// TIA Portal project "Smart-greenhouse" (V16)

(* hardware
DEVICE "S7-1200 station_1"  S7-1200 Station
   slot 0: "Telaio di montaggio_0"  S7-1200 Rack  Rack  V1.0
   slot 1: "PLC_1"  CPU 1212C AC/DC/Rly  6ES7 212-1BE40-0XB0  V4.4
*)

// ===== PLC "PLC_1"  CPU 1212C AC/DC/Rly =====

VAR_GLOBAL   // PLC tag table "Tabella delle variabili standard"
   "GripperOpenStop" AT %I0.0 : Bool;
   "GripperCounter" AT %I0.1 : Bool;
   "ArmBackStop" AT %I0.2 : Bool;
   "ArmHCounter" AT %I0.3 : Bool;
   "ArmTopStop" AT %I0.4 : Bool;
   "ArmRotationStop" AT %I0.5 : Bool;
   "RotationalEncoder" AT %ID1000 : DInt;
   "VerticalEncoder" AT %ID1004 : DInt;
   "ConnectionButton" AT %I1.2 : Bool;
   "StopButton" AT %I1.3 : Bool;
   "ResetButton" AT %I1.4 : Bool;
   "Photosensor" AT %I1.5 : Bool;
   "GripperOpen" AT %Q0.0 : Bool;
   "GripperClose" AT %Q0.1 : Bool;
   "ArmFront" AT %Q0.2 : Bool;
   "ArmBack" AT %Q0.3 : Bool;
   "ArmDown" AT %Q0.4 : Bool;
   "ArmUp" AT %Q0.5 : Bool;
   "RotationClockwise" AT %Q0.6 : Bool;
   "RotationCounterclockwise" AT %Q0.7 : Bool;
   "GreenLed" AT %Q1.0 : Bool;
   "StopConveyor" AT %Q1.1 : Bool;
   "System_Byte" AT %MB1 : Byte;
   "FirstScan" AT %M6.0 : Bool;
   "DiagStatusUpdate" AT %M6.1 : Bool;
   "AlwaysTRUE" AT %M6.2 : Bool;
   "AlwaysFALSE" AT %M6.3 : Bool;
   "RotationalCounter" AT %MW2 : UInt;
   "Clock_Byte" AT %MB0 : Byte;
   "Clock_10Hz" AT %M0.0 : Bool;
   "Clock_5Hz" AT %M0.1 : Bool;
   "Clock_2.5Hz" AT %M0.2 : Bool;
   "Clock_2Hz" AT %M0.3 : Bool;
   "Clock_1.25Hz" AT %M0.4 : Bool;
   "Clock_1Hz" AT %M0.5 : Bool;
   "Clock_0.625Hz" AT %M0.6 : Bool;
   "Clock_0.5Hz" AT %M0.7 : Bool;
   "VerticalCounter" AT %MW4 : UInt;
   "ForceReset" AT %M7.0 : Bool;
   "ResetCompleted" AT %M7.1 : Bool;
   "TCON_Req" AT %M1.0 : Bool;
   "TDIS_Req" AT %M1.1 : Bool;
   "TSEND_Req" AT %M1.2 : Bool;
   "TRCV_Req" AT %M1.3 : Bool;
   "VerticalOverCounter" AT %MW8 : Int;
   "VerticalUnderCounter" AT %MW10 : Int;
   "RotationOverCounter" AT %MW12 : Int;
   "RotationUnderCounter" AT %MW14 : Int;
   "NormalizedRotationUnderCounter" AT %MW16 : Int;
   "NormalizedVerticalUnderCounter" AT %MW18 : Int;
   "StopAll" AT %M20.1 : Bool;
   "HRegistered" AT %M20.2 : Bool;
   "RRegistered" AT %M20.3 : Bool;
   "VRegistered" AT %M20.4 : Bool;
   "State 0" AT %M20.5 : Bool;
   "State 3" AT %M20.6 : Bool;
   "AuxPhotocellStatus" AT %M20.7 : Bool;
   "State 3.1" AT %M21.0 : Bool;
   "State 3.2" AT %M21.1 : Bool;
   "HallEffectSensor" AT %I1.6 : Bool;
   "Sprinkler" AT %Q1.2 : Bool;
   "ArmTriggerOut_REQ" AT %M21.2 : Bool;
   "Test" AT %M21.3 : Bool;
   "MotorOn" AT %M21.4 : Bool;
   "TESTSOCKET" AT %M21.5 : Bool;
   "ForceMotor" AT %M21.6 : Bool;
   "AuxStop" AT %M21.7 : Bool;
   "State 3.1.1" AT %M22.0 : Bool;
   "State 3.1.2" AT %M22.1 : Bool;
   "State 3.1.3" AT %M22.2 : Bool;
   "State 3.3" AT %M22.3 : Bool;
   "State 1" AT %M22.4 : Bool;
   "State 1.1" AT %M22.5 : Bool;
   "State 1.2" AT %M22.6 : Bool;
   "State 1.3" AT %M22.7 : Bool;
   "State 2" AT %M23.0 : Bool;
   "AuxLapNotCompleted" AT %M23.1 : Bool;
   "HighTemp" AT %I1.7 : Bool;
   "LowTemp" AT %I2.0 : Bool;
   "HighHum" AT %I2.1 : Bool;
   "AuxHighTemp" AT %M23.2 : Bool;
   "AuxLowTemp" AT %M23.3 : Bool;
   "AuxHum" AT %M23.4 : Bool;
   "WindowPiston" AT %Q1.3 : Bool;
   "IRLamp" AT %Q1.4 : Bool;
   "Fan" AT %Q1.5 : Bool;
   "Tag_1" AT %MW0 : Int;
END_VAR

DATA_BLOCK "REAL TIME DATA"   // DB4
{ S7_Optimized_Access := 'TRUE' }
VERSION : 0.1
   VAR
      "REAL TIME DATA" : DTL;
   END_VAR
BEGIN
END_DATA_BLOCK

DATA_BLOCK "Trigger_values"   // DB7
{ S7_Optimized_Access := 'FALSE' }
VERSION : 0.1
   VAR
      Trigger : Bool;
   END_VAR
BEGIN
END_DATA_BLOCK

DATA_BLOCK "Sent_values"   // DB10
{ S7_Optimized_Access := 'FALSE' }
VERSION : 0.1
   VAR
      Rotation : Int;
      Vertical : Int;
      Horizontal : Int;
      Gripper : Bool;
   END_VAR
BEGIN
END_DATA_BLOCK

DATA_BLOCK "Received_values"   // DB12
{ S7_Optimized_Access := 'FALSE' }
VERSION : 0.1
   VAR
      Rotation : Int;
      Vertical : Int;
      Horizontal : Int;
      Gripper : Bool;
   END_VAR
BEGIN
END_DATA_BLOCK

DATA_BLOCK "Obj_detect"   // DB20
{ S7_Optimized_Access := 'FALSE' }
VERSION : 0.1
   VAR
      message : String := 'START';
   END_VAR
BEGIN
END_DATA_BLOCK

// folder: System blocks/Program resources

DATA_BLOCK "CONTATORE"   // DB1
{ S7_Optimized_Access := 'TRUE' }
AUTHOR : Simatic
FAMILY : IEC
NAME : CNTR
VERSION : 1.0
// stored: InstanceOfName IEC_COUNTER
"IEC_COUNTER"
BEGIN
END_DATA_BLOCK

DATA_BLOCK "Timer Sprinkler"   // DB2
{ S7_Optimized_Access := 'TRUE' }
AUTHOR : Simatic
FAMILY : IEC
NAME : IEC_TMR
VERSION : 1.0
// stored: InstanceOfName IEC_TIMER
"IEC_TIMER"
BEGIN
END_DATA_BLOCK

DATA_BLOCK "ArmHCounterCTUD"   // DB3
{ S7_Optimized_Access := 'TRUE' }
AUTHOR : Simatic
FAMILY : IEC
NAME : CNTR
VERSION : 1.0
// stored: InstanceOfName IEC_COUNTER
"IEC_COUNTER"
BEGIN
END_DATA_BLOCK

DATA_BLOCK "PLC_1_Connection_DB"   // DB6
{ S7_Optimized_Access := 'TRUE' }
AUTHOR : SIMATIC
FAMILY : MC7Plus
NAME : TC_IP_v4
VERSION : 1.0
// stored: InstanceOfName TCON_IP_v4
"TCON_IP_v4"
BEGIN
   ID := 1;
   InterfaceId := 64;
   RemotePort := 2001;
   ActiveEstablished := true;
   RemoteAddress.ADDR[1] := 192;
   RemoteAddress.ADDR[2] := 168;
   RemoteAddress.ADDR[4] := 9;
END_DATA_BLOCK

DATA_BLOCK "ArmHStatusCTUD"   // DB9
{ S7_Optimized_Access := 'TRUE' }
AUTHOR : Simatic
FAMILY : IEC
NAME : CNTR
VERSION : 1.0
// stored: InstanceOfName IEC_COUNTER
"IEC_COUNTER"
BEGIN
END_DATA_BLOCK

DATA_BLOCK "GripperStatus"   // DB15
{ S7_Optimized_Access := 'TRUE' }
AUTHOR : Simatic
FAMILY : IEC
NAME : CNTR
VERSION : 1.0
// stored: InstanceOfName IEC_COUNTER
"IEC_COUNTER"
BEGIN
END_DATA_BLOCK

DATA_BLOCK "ArmHStatus"   // DB16
{ S7_Optimized_Access := 'TRUE' }
AUTHOR : Simatic
FAMILY : IEC
NAME : CNTR
VERSION : 1.0
// stored: InstanceOfName IEC_COUNTER
"IEC_COUNTER"
BEGIN
END_DATA_BLOCK

DATA_BLOCK "IEC_Timer_0_DB"   // DB17
{ S7_Optimized_Access := 'TRUE' }
AUTHOR : Simatic
FAMILY : IEC
NAME : IEC_TMR
VERSION : 1.0
// stored: InstanceOfName IEC_TIMER
"IEC_TIMER"
BEGIN
END_DATA_BLOCK

DATA_BLOCK "IEC_Timer_0_DB_1"   // DB18
{ S7_Optimized_Access := 'TRUE' }
AUTHOR : Simatic
FAMILY : IEC
NAME : IEC_TMR
VERSION : 1.0
// stored: InstanceOfName IEC_TIMER
"IEC_TIMER"
BEGIN
END_DATA_BLOCK

// folder: (top level)

ORGANIZATION_BLOCK "Main"   // OB1, LAD, ProgramCycle
TITLE = "Main Program Sweep (Cycle)"
{ S7_Optimized_Access := 'TRUE' }
VERSION : 0.1
   VAR_INPUT
      Initial_Call : Bool;   // Initial call of this OB
      Remanence : Bool;   // =True, if remanent data are available
   END_VAR
   VAR_TEMP   // added for the SCL form of the ladder/FBD networks
      _w1 : Bool;
      _w2 : Bool;
      _w3 : Bool;
      _w4 : Bool;
      _w5 : Bool;
      _w6 : Bool;
      _w7 : Bool;
   END_VAR
BEGIN

REGION Network 1: State inizialization
   // All'avvio del PLC vengono inizializzati gli stati
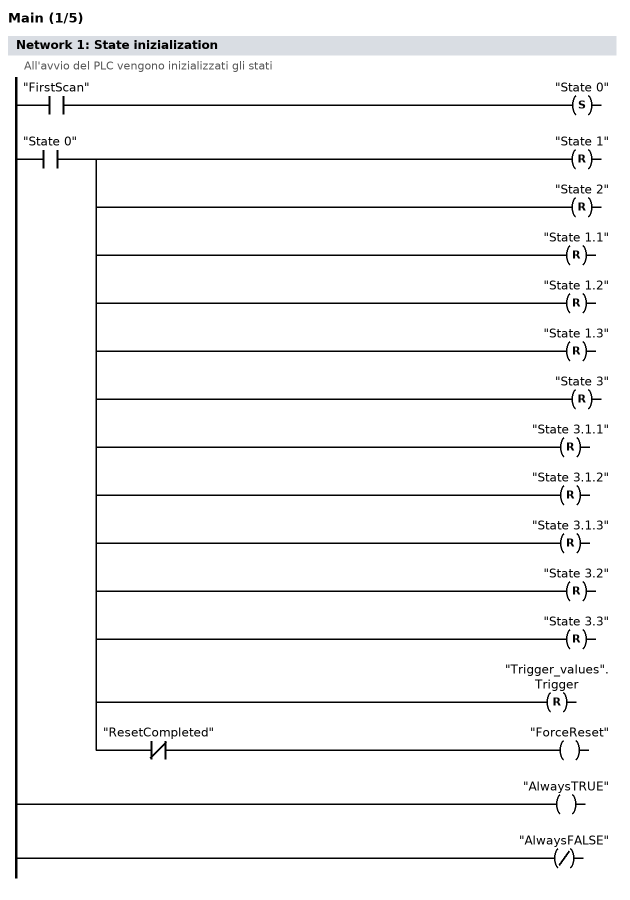
   RUNG wire#powerrail
      Contact( "FirstScan" )
      S_Coil( "State 0" )
   END_RUNG
   RUNG wire#powerrail
      Contact( "State 0" )
      wire#w1
      R_Coil( "State 1" )
   END_RUNG
   RUNG wire#w1
      R_Coil( "State 2" )
   END_RUNG
   RUNG wire#w1
      R_Coil( "State 1.1" )
   END_RUNG
   RUNG wire#w1
      R_Coil( "State 1.2" )
   END_RUNG
   RUNG wire#w1
      R_Coil( "State 1.3" )
   END_RUNG
   RUNG wire#w1
      R_Coil( "State 3" )
   END_RUNG
   RUNG wire#w1
      R_Coil( "State 3.1.1" )
   END_RUNG
   RUNG wire#w1
      R_Coil( "State 3.1.2" )
   END_RUNG
   RUNG wire#w1
      R_Coil( "State 3.1.3" )
   END_RUNG
   RUNG wire#w1
      R_Coil( "State 3.2" )
   END_RUNG
   RUNG wire#w1
      R_Coil( "State 3.3" )
   END_RUNG
   RUNG wire#w1
      R_Coil( "Trigger_values".Trigger )
   END_RUNG
   RUNG wire#w1
      I_Contact( "ResetCompleted" )
      Coil( "ForceReset" )
   END_RUNG
   RUNG wire#powerrail
      Coil( "AlwaysTRUE" )
   END_RUNG
   RUNG wire#powerrail
      I_Coil( "AlwaysFALSE" )
   END_RUNG
   // the same network as SCL:
   IF "FirstScan" THEN "State 0" := TRUE; END_IF;
   IF "State 0" THEN
       "State 1" := FALSE;
       "State 2" := FALSE;
       "State 1.1" := FALSE;
       "State 1.2" := FALSE;
       "State 1.3" := FALSE;
       "State 3" := FALSE;
       "State 3.1.1" := FALSE;
       "State 3.1.2" := FALSE;
       "State 3.1.3" := FALSE;
       "State 3.2" := FALSE;
       "State 3.3" := FALSE;
       "Trigger_values".Trigger := FALSE;
   END_IF;
   "ForceReset" := "State 0" AND NOT "ResetCompleted";
   "AlwaysTRUE" := TRUE;
   "AlwaysFALSE" := NOT TRUE;
END_REGION

REGION Network 2: Gestione braccio robotico
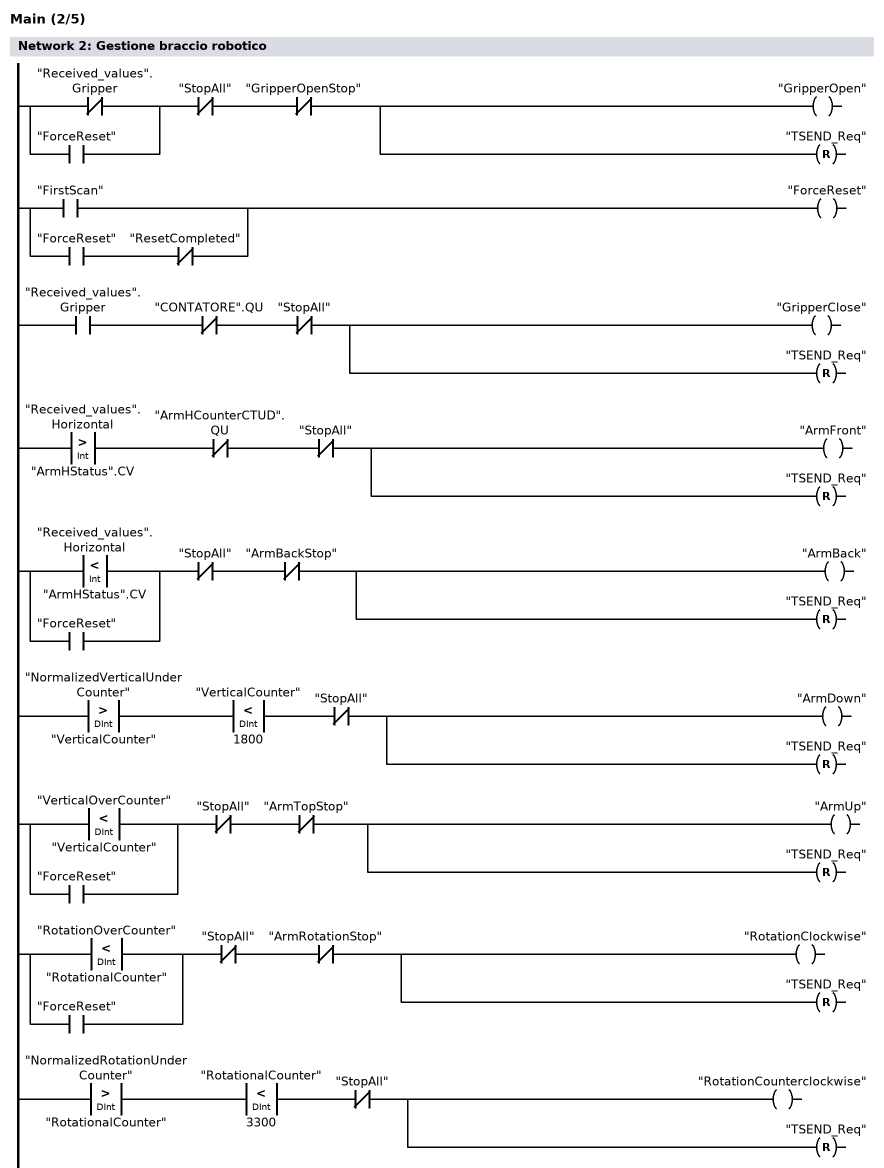
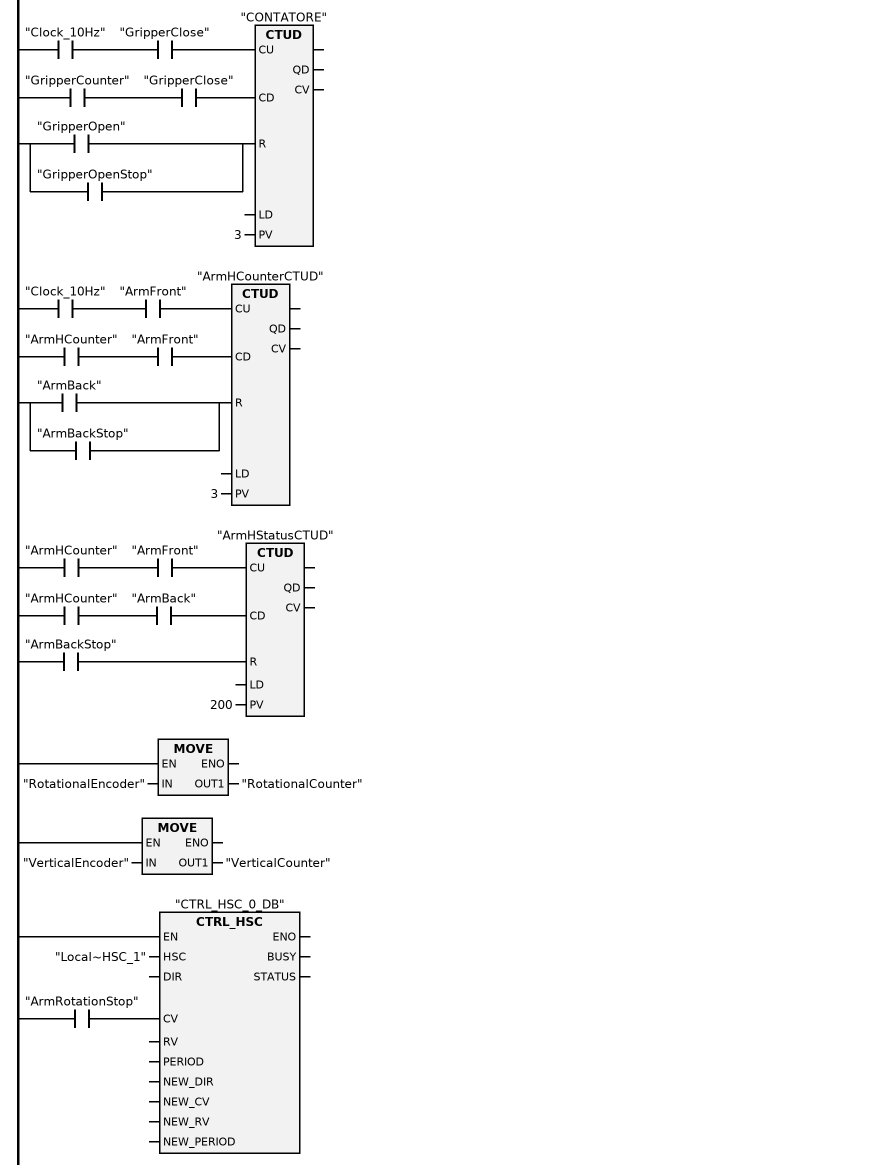
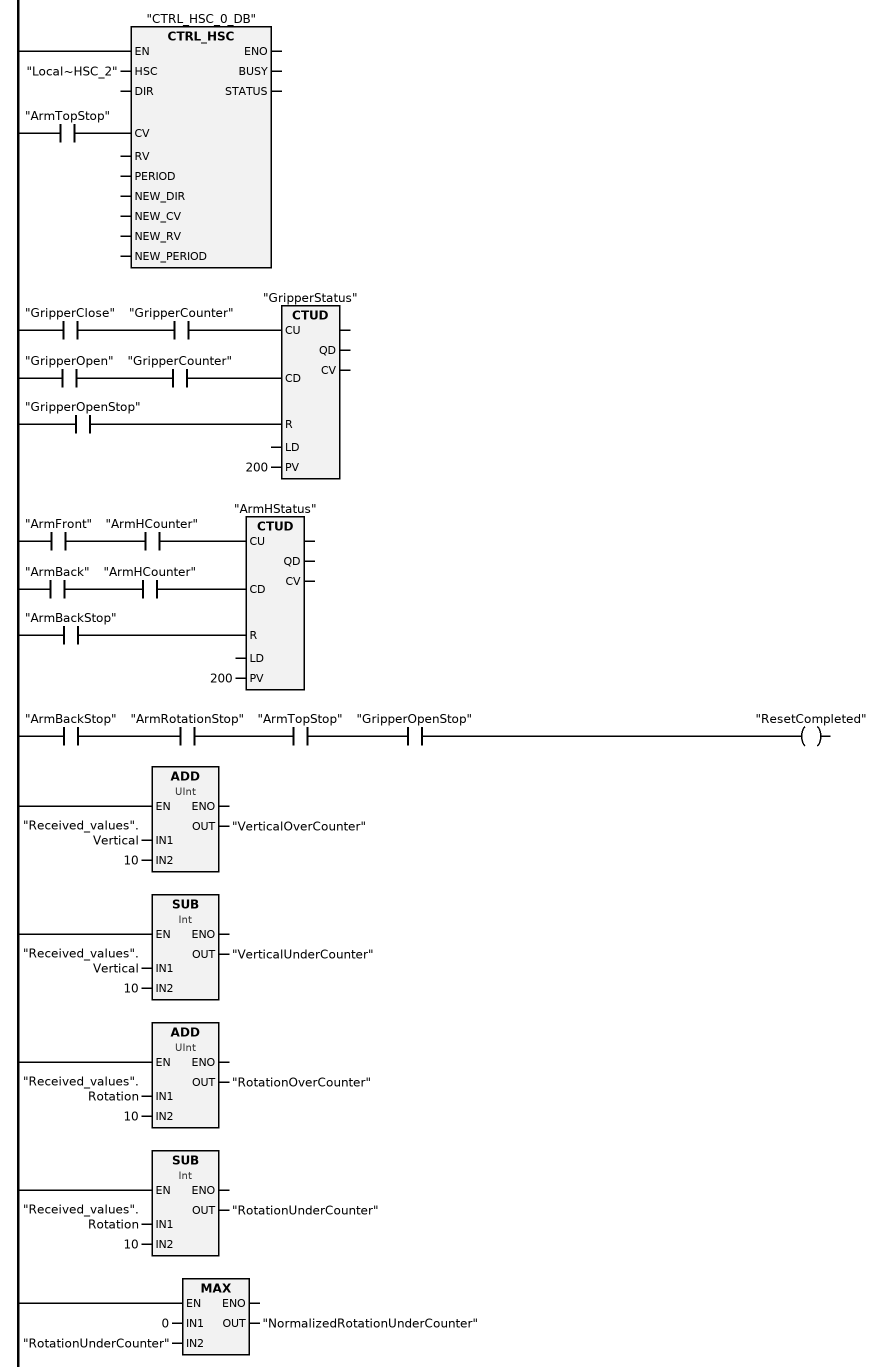
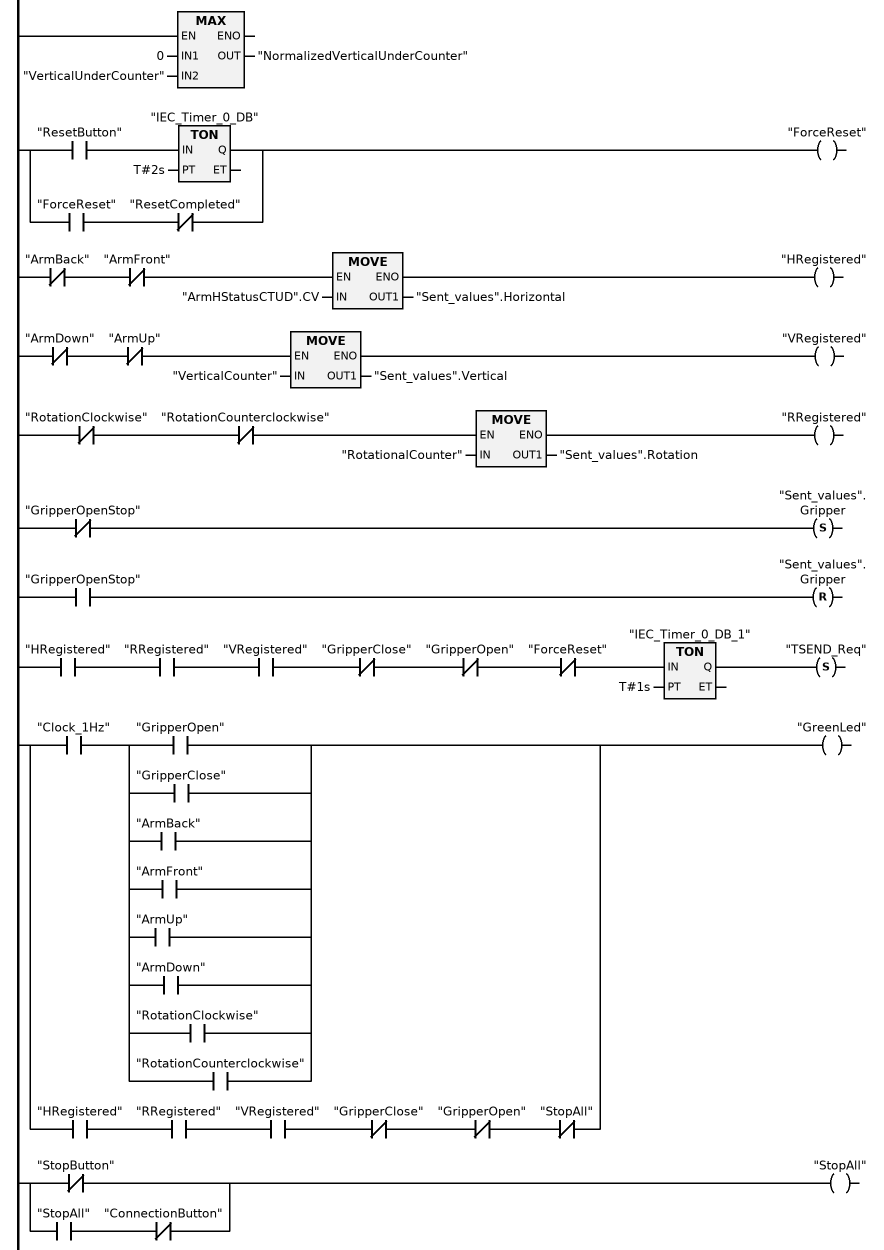
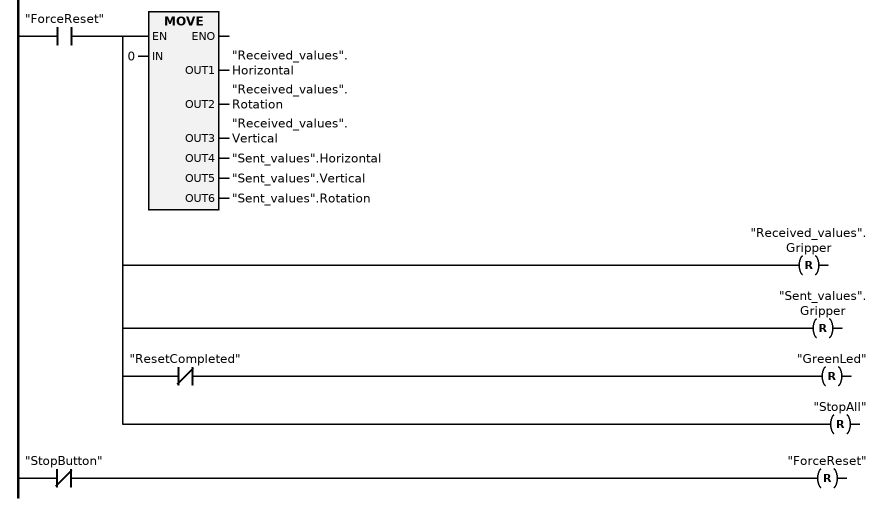
   "GripperOpen" := (NOT "Received_values".Gripper OR "ForceReset") AND NOT "StopAll" AND NOT "GripperOpenStop";
   IF "GripperOpen" THEN "TSEND_Req" := FALSE; END_IF;
   "ForceReset" := "FirstScan" OR ("ForceReset" AND NOT "ResetCompleted");
   "GripperClose" := "Received_values".Gripper AND NOT "CONTATORE".QU AND NOT "StopAll";
   IF "GripperClose" THEN "TSEND_Req" := FALSE; END_IF;
   "ArmFront" := ("Received_values".Horizontal > "ArmHStatus".CV) AND NOT "ArmHCounterCTUD".QU AND NOT "StopAll";
   IF "ArmFront" THEN "TSEND_Req" := FALSE; END_IF;
   "ArmBack" := (("Received_values".Horizontal < "ArmHStatus".CV) OR "ForceReset") AND NOT "StopAll" AND NOT "ArmBackStop";
   IF "ArmBack" THEN "TSEND_Req" := FALSE; END_IF;
   "ArmDown" := ("NormalizedVerticalUnderCounter" > "VerticalCounter") AND ("VerticalCounter" < 1800) AND NOT "StopAll";
   IF "ArmDown" THEN "TSEND_Req" := FALSE; END_IF;
   "ArmUp" := (("VerticalOverCounter" < "VerticalCounter") OR "ForceReset") AND NOT "StopAll" AND NOT "ArmTopStop";
   IF "ArmUp" THEN "TSEND_Req" := FALSE; END_IF;
   "RotationClockwise" := (("RotationOverCounter" < "RotationalCounter") OR "ForceReset") AND NOT "StopAll" AND NOT "ArmRotationStop";
   IF "RotationClockwise" THEN "TSEND_Req" := FALSE; END_IF;
   "RotationCounterclockwise" := ("NormalizedRotationUnderCounter" > "RotationalCounter") AND ("RotationalCounter" < 3300) AND NOT "StopAll";
   IF "RotationCounterclockwise" THEN "TSEND_Req" := FALSE; END_IF;
   "CONTATORE".CTUD(CU := "Clock_10Hz" AND "GripperClose",
                    CD := "GripperCounter" AND "GripperClose",
                    R := "GripperOpen" OR "GripperOpenStop",
                    PV := 3);
   "ArmHCounterCTUD".CTUD(CU := "Clock_10Hz" AND "ArmFront",
                          CD := "ArmHCounter" AND "ArmFront",
                          R := "ArmBack" OR "ArmBackStop",
                          PV := 3);
   "ArmHStatusCTUD".CTUD(CU := "ArmHCounter" AND "ArmFront",
                         CD := "ArmHCounter" AND "ArmBack",
                         R := "ArmBackStop",
                         PV := 200);
   "RotationalCounter" := "RotationalEncoder";
   "VerticalCounter" := "VerticalEncoder";
   "CTRL_HSC_0_DB"(HSC := "Local~HSC_1", CV := "ArmRotationStop");   // CTRL_HSC
   "CTRL_HSC_0_DB"(HSC := "Local~HSC_2", CV := "ArmTopStop");   // CTRL_HSC
   "GripperStatus".CTUD(CU := "GripperClose" AND "GripperCounter",
                        CD := "GripperOpen" AND "GripperCounter",
                        R := "GripperOpenStop",
                        PV := 200);
   "ArmHStatus".CTUD(CU := "ArmFront" AND "ArmHCounter",
                     CD := "ArmBack" AND "ArmHCounter",
                     R := "ArmBackStop",
                     PV := 200);
   "ResetCompleted" := "ArmBackStop" AND "ArmRotationStop" AND "ArmTopStop" AND "GripperOpenStop";
   "VerticalOverCounter" := "Received_values".Vertical + 10;
   "VerticalUnderCounter" := "Received_values".Vertical - 10;
   "RotationOverCounter" := "Received_values".Rotation + 10;
   "RotationUnderCounter" := "Received_values".Rotation - 10;
   "NormalizedRotationUnderCounter" := MAX(IN1 := 0, IN2 := "RotationUnderCounter");
   "NormalizedVerticalUnderCounter" := MAX(IN1 := 0, IN2 := "VerticalUnderCounter");
   "IEC_Timer_0_DB".TON(IN := "ResetButton", PT := T#2s);
   "ForceReset" := "IEC_Timer_0_DB".Q OR ("ForceReset" AND NOT "ResetCompleted");
   #_w1 := NOT "ArmBack" AND NOT "ArmFront";
   IF #_w1 THEN "Sent_values".Horizontal := "ArmHStatusCTUD".CV; END_IF;
   "HRegistered" := #_w1;
   #_w2 := NOT "ArmDown" AND NOT "ArmUp";
   IF #_w2 THEN "Sent_values".Vertical := "VerticalCounter"; END_IF;
   "VRegistered" := #_w2;
   #_w3 := NOT "RotationClockwise" AND NOT "RotationCounterclockwise";
   IF #_w3 THEN "Sent_values".Rotation := "RotationalCounter"; END_IF;
   "RRegistered" := #_w3;
   IF NOT "GripperOpenStop" THEN "Sent_values".Gripper := TRUE; END_IF;
   IF "GripperOpenStop" THEN "Sent_values".Gripper := FALSE; END_IF;
   "IEC_Timer_0_DB_1".TON(IN := "HRegistered" AND "RRegistered" AND "VRegistered" AND NOT "GripperClose" AND NOT "GripperOpen" AND NOT "ForceReset",
                          PT := T#1s);
   IF "IEC_Timer_0_DB_1".Q THEN "TSEND_Req" := TRUE; END_IF;
   "GreenLed" := ("Clock_1Hz" AND ("GripperOpen" OR "GripperClose" OR "ArmBack" OR "ArmFront" OR "ArmUp" OR "ArmDown" OR "RotationClockwise" OR "RotationCounterclockwise")) OR ("HRegistered" AND "RRegistered" AND "VRegistered" AND NOT "GripperClose" AND NOT "GripperOpen" AND NOT "StopAll");
   "StopAll" := NOT "StopButton" OR ("StopAll" AND NOT "ConnectionButton");
   IF "ForceReset" THEN
       "Received_values".Horizontal := 0;
       "Received_values".Rotation := 0;
       "Received_values".Vertical := 0;
       "Sent_values".Horizontal := 0;
       "Sent_values".Vertical := 0;
       "Sent_values".Rotation := 0;
       "Received_values".Gripper := FALSE;
       "Sent_values".Gripper := FALSE;
   END_IF;
   IF "ForceReset" AND NOT "ResetCompleted" THEN "GreenLed" := FALSE; END_IF;
   IF "ForceReset" THEN "StopAll" := FALSE; END_IF;
   IF NOT "StopButton" THEN "ForceReset" := FALSE; END_IF;
END_REGION

REGION Network 3: RESET
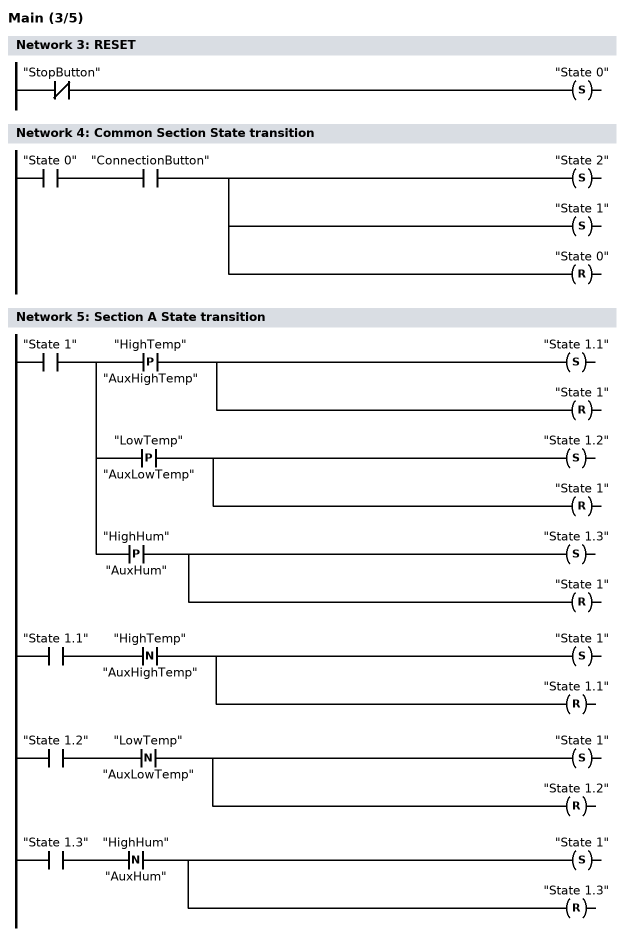
   RUNG wire#powerrail
      I_Contact( "StopButton" )
      S_Coil( "State 0" )
   END_RUNG
   // the same network as SCL:
   IF NOT "StopButton" THEN "State 0" := TRUE; END_IF;
END_REGION

REGION Network 4: Common Section State transition
   RUNG wire#powerrail
      Contact( "State 0" )
      Contact( "ConnectionButton" )
      wire#w1
      S_Coil( "State 2" )
   END_RUNG
   RUNG wire#w1
      S_Coil( "State 1" )
   END_RUNG
   RUNG wire#w1
      R_Coil( "State 0" )
   END_RUNG
   // the same network as SCL:
   IF "State 0" AND "ConnectionButton" THEN
       "State 2" := TRUE;
       "State 1" := TRUE;
       "State 0" := FALSE;
   END_IF;
END_REGION

REGION Network 5: Section A State transition
   RUNG wire#powerrail
      Contact( "State 1" )
      wire#w1
      P_Contact(operand := "HighTemp", bit := "AuxHighTemp")
      wire#w2
      S_Coil( "State 1.1" )
   END_RUNG
   RUNG wire#w2
      R_Coil( "State 1" )
   END_RUNG
   RUNG wire#w1
      P_Contact(operand := "LowTemp", bit := "AuxLowTemp")
      wire#w3
      S_Coil( "State 1.2" )
   END_RUNG
   RUNG wire#w3
      R_Coil( "State 1" )
   END_RUNG
   RUNG wire#w1
      P_Contact(operand := "HighHum", bit := "AuxHum")
      wire#w4
      S_Coil( "State 1.3" )
   END_RUNG
   RUNG wire#w4
      R_Coil( "State 1" )
   END_RUNG
   RUNG wire#powerrail
      Contact( "State 1.1" )
      N_Contact(operand := "HighTemp", bit := "AuxHighTemp")
      wire#w5
      S_Coil( "State 1" )
   END_RUNG
   RUNG wire#w5
      R_Coil( "State 1.1" )
   END_RUNG
   RUNG wire#powerrail
      Contact( "State 1.2" )
      N_Contact(operand := "LowTemp", bit := "AuxLowTemp")
      wire#w6
      S_Coil( "State 1" )
   END_RUNG
   RUNG wire#w6
      R_Coil( "State 1.2" )
   END_RUNG
   RUNG wire#powerrail
      Contact( "State 1.3" )
      N_Contact(operand := "HighHum", bit := "AuxHum")
      wire#w7
      S_Coil( "State 1" )
   END_RUNG
   RUNG wire#w7
      R_Coil( "State 1.3" )
   END_RUNG
   // the same network as SCL:
   #_w1 := "State 1" AND "HighTemp" AND NOT "AuxHighTemp";   // rising edge of "HighTemp"
   "AuxHighTemp" := "HighTemp";
   IF #_w1 THEN "State 1.1" := TRUE; END_IF;
   #_w2 := "State 1";
   IF #_w1 THEN "State 1" := FALSE; END_IF;
   #_w3 := #_w2 AND "LowTemp" AND NOT "AuxLowTemp";   // rising edge of "LowTemp"
   "AuxLowTemp" := "LowTemp";
   IF #_w3 THEN
       "State 1.2" := TRUE;
       "State 1" := FALSE;
   END_IF;
   #_w4 := #_w2 AND "HighHum" AND NOT "AuxHum";   // rising edge of "HighHum"
   "AuxHum" := "HighHum";
   IF #_w4 THEN
       "State 1.3" := TRUE;
       "State 1" := FALSE;
   END_IF;
   #_w5 := "State 1.1" AND NOT "HighTemp" AND "AuxHighTemp";   // falling edge of "HighTemp"
   "AuxHighTemp" := "HighTemp";
   IF #_w5 THEN
       "State 1" := TRUE;
       "State 1.1" := FALSE;
   END_IF;
   #_w6 := "State 1.2" AND NOT "LowTemp" AND "AuxLowTemp";   // falling edge of "LowTemp"
   "AuxLowTemp" := "LowTemp";
   IF #_w6 THEN
       "State 1" := TRUE;
       "State 1.2" := FALSE;
   END_IF;
   #_w7 := "State 1.3" AND NOT "HighHum" AND "AuxHum";   // falling edge of "HighHum"
   "AuxHum" := "HighHum";
   IF #_w7 THEN
       "State 1" := TRUE;
       "State 1.3" := FALSE;
   END_IF;
END_REGION

REGION Network 6: Section B State transition
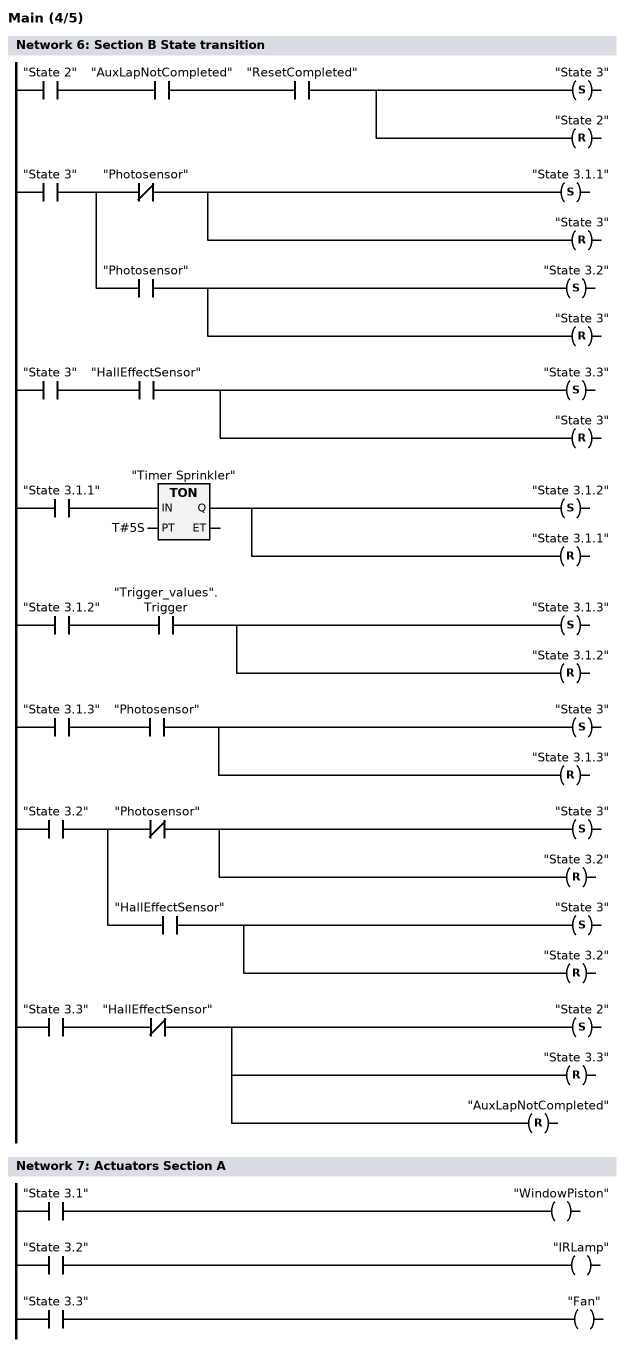
   IF "State 2" AND "AuxLapNotCompleted" AND "ResetCompleted" THEN
       "State 3" := TRUE;
       "State 2" := FALSE;
   END_IF;
   IF "State 3" AND NOT "Photosensor" THEN "State 3.1.1" := TRUE; END_IF;
   #_w1 := "State 3";
   IF "State 3" AND NOT "Photosensor" THEN "State 3" := FALSE; END_IF;
   IF #_w1 AND "Photosensor" THEN
       "State 3.2" := TRUE;
       "State 3" := FALSE;
   END_IF;
   IF "State 3" AND "HallEffectSensor" THEN
       "State 3.3" := TRUE;
       "State 3" := FALSE;
   END_IF;
   "Timer Sprinkler".TON(IN := "State 3.1.1", PT := T#5S);
   IF "Timer Sprinkler".Q THEN
       "State 3.1.2" := TRUE;
       "State 3.1.1" := FALSE;
   END_IF;
   IF "State 3.1.2" AND "Trigger_values".Trigger THEN
       "State 3.1.3" := TRUE;
       "State 3.1.2" := FALSE;
   END_IF;
   IF "State 3.1.3" AND "Photosensor" THEN
       "State 3" := TRUE;
       "State 3.1.3" := FALSE;
   END_IF;
   IF "State 3.2" AND NOT "Photosensor" THEN "State 3" := TRUE; END_IF;
   #_w2 := "State 3.2";
   IF "State 3.2" AND NOT "Photosensor" THEN "State 3.2" := FALSE; END_IF;
   IF #_w2 AND "HallEffectSensor" THEN
       "State 3" := TRUE;
       "State 3.2" := FALSE;
   END_IF;
   IF "State 3.3" AND NOT "HallEffectSensor" THEN "State 2" := TRUE; END_IF;
   #_w3 := "State 3.3" AND NOT "HallEffectSensor";
   IF #_w3 THEN
       "State 3.3" := FALSE;
       "AuxLapNotCompleted" := FALSE;
   END_IF;
END_REGION

REGION Network 7: Actuators Section A
   RUNG wire#powerrail
      Contact( "State 3.1" )
      Coil( "WindowPiston" )
   END_RUNG
   RUNG wire#powerrail
      Contact( "State 3.2" )
      Coil( "IRLamp" )
   END_RUNG
   RUNG wire#powerrail
      Contact( "State 3.3" )
      Coil( "Fan" )
   END_RUNG
   // the same network as SCL:
   "WindowPiston" := "State 3.1";
   "IRLamp" := "State 3.2";
   "Fan" := "State 3.3";
END_REGION

REGION Network 8: Actuators Section B
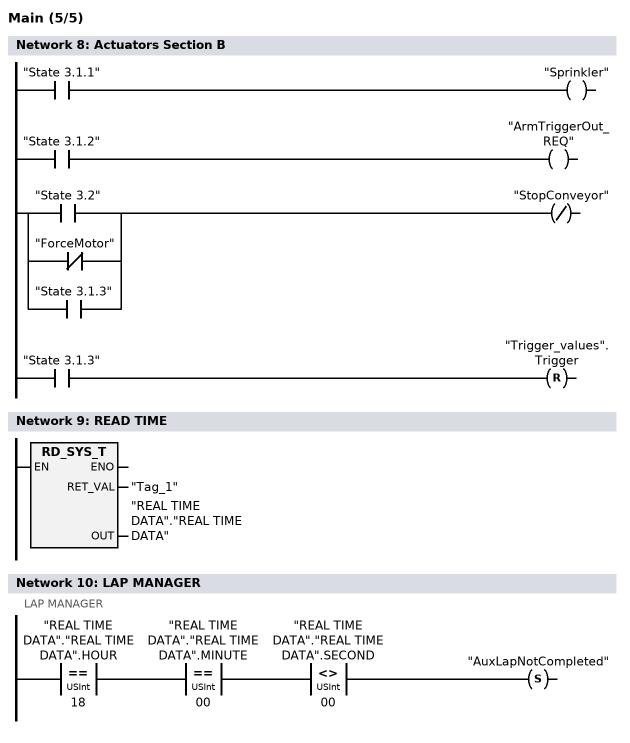
   RUNG wire#powerrail
      Contact( "State 3.1.1" )
      Coil( "Sprinkler" )
   END_RUNG
   RUNG wire#powerrail
      Contact( "State 3.1.2" )
      Coil( "ArmTriggerOut_REQ" )
   END_RUNG
   RUNG wire#powerrail
      Contact( "State 3.2" )
      wire#w1
      I_Coil( "StopConveyor" )
   END_RUNG
   RUNG wire#powerrail
      I_Contact( "ForceMotor" )
   END_RUNG wire#w1
   RUNG wire#powerrail
      Contact( "State 3.1.3" )
   END_RUNG wire#w1
   RUNG wire#powerrail
      Contact( "State 3.1.3" )
      R_Coil( "Trigger_values".Trigger )
   END_RUNG
   // the same network as SCL:
   "Sprinkler" := "State 3.1.1";
   "ArmTriggerOut_REQ" := "State 3.1.2";
   "StopConveyor" := NOT ("State 3.2" OR NOT "ForceMotor" OR "State 3.1.3");
   IF "State 3.1.3" THEN "Trigger_values".Trigger := FALSE; END_IF;
END_REGION

REGION Network 9: READ TIME
   "Tag_1" := RD_SYS_T(OUT => "REAL TIME DATA"."REAL TIME DATA");
END_REGION

REGION Network 10: LAP MANAGER
   // LAP MANAGER
   RUNG wire#powerrail
      { S7_Templates := "SrcType := USInt" } EQ_Contact(in1 := "REAL TIME DATA"."REAL TIME DATA".HOUR, in2 := 18)
      { S7_Templates := "SrcType := USInt" } EQ_Contact(in1 := "REAL TIME DATA"."REAL TIME DATA".MINUTE, in2 := 00)
      { S7_Templates := "SrcType := USInt" } NE_Contact(in1 := "REAL TIME DATA"."REAL TIME DATA".SECOND, in2 := 00)
      S_Coil( "AuxLapNotCompleted" )
   END_RUNG
   // the same network as SCL:
   IF ("REAL TIME DATA"."REAL TIME DATA".HOUR = 18) AND ("REAL TIME DATA"."REAL TIME DATA".MINUTE = 00) AND ("REAL TIME DATA"."REAL TIME DATA".SECOND <> 00) THEN
       "AuxLapNotCompleted" := TRUE;
   END_IF;
END_REGION
END_ORGANIZATION_BLOCK